(* CoDeSys 2.3 export: LogDInt.EXP *)

(* POU basic/LogDInt, ST *)
FUNCTION LogDInt : BOOL
VAR_INPUT
    Group: BYTE;
    Id: BYTE;
    Channel: UINT;
    Value: DINT;
END_VAR
VAR
END_VAR
IF Group > 0 OR Id > 0 THEN
    IF Channel < 256 THEN
        EvtGr8Id8Ch8Tick32Int32(Group, Id, UINT_TO_BYTE(Channel), GlobalTick, Value, GlobalLogBufferHandle);
    ELSE
        EvtGr8Id8Ch16Tick32Int32(Group, Id, Channel, GlobalTick, Value, GlobalLogBufferHandle);
    END_IF
ELSIF Channel < 256 THEN
    EvtCh8Tick32Int32(UINT_TO_BYTE(Channel), GlobalTick, Value, GlobalLogBufferHandle);
ELSE
    EvtCh16Tick32Int32(Channel, GlobalTick, Value, GlobalLogBufferHandle);
END_IF
END_FUNCTION
